PROGRAM Callblocks
VAR
	
CC1_Clamp_Unit1_3 : clamp;
CC2_Clamp_Unit2_3 : clamp;
CC3_Clamp_Unit3_3 : clamp;
CC4_Clamp_Unit4_3 : clamp;
CC5_Clamp_Unit5_1 : clamp;
CC6_Clamp_Unit6_1 : clamp;

Temp_bool : BOOL;
Feedback_Unit1  : Feedback_FB;
Feedback_Unit2  : Feedback_FB;
Feedback_Unit3  : Feedback_FB;
Feedback_Unit4  : Feedback_FB;
Feedback_Unit5  : Feedback_FB;
Feedback_Unit6  : Feedback_FB;


Door           : RollerDoor;
Trunion        : Trunion;
TT             : Turntable ;
Robot1         : Weldrobot;
Robot2         : MHrobot;

END_VAR

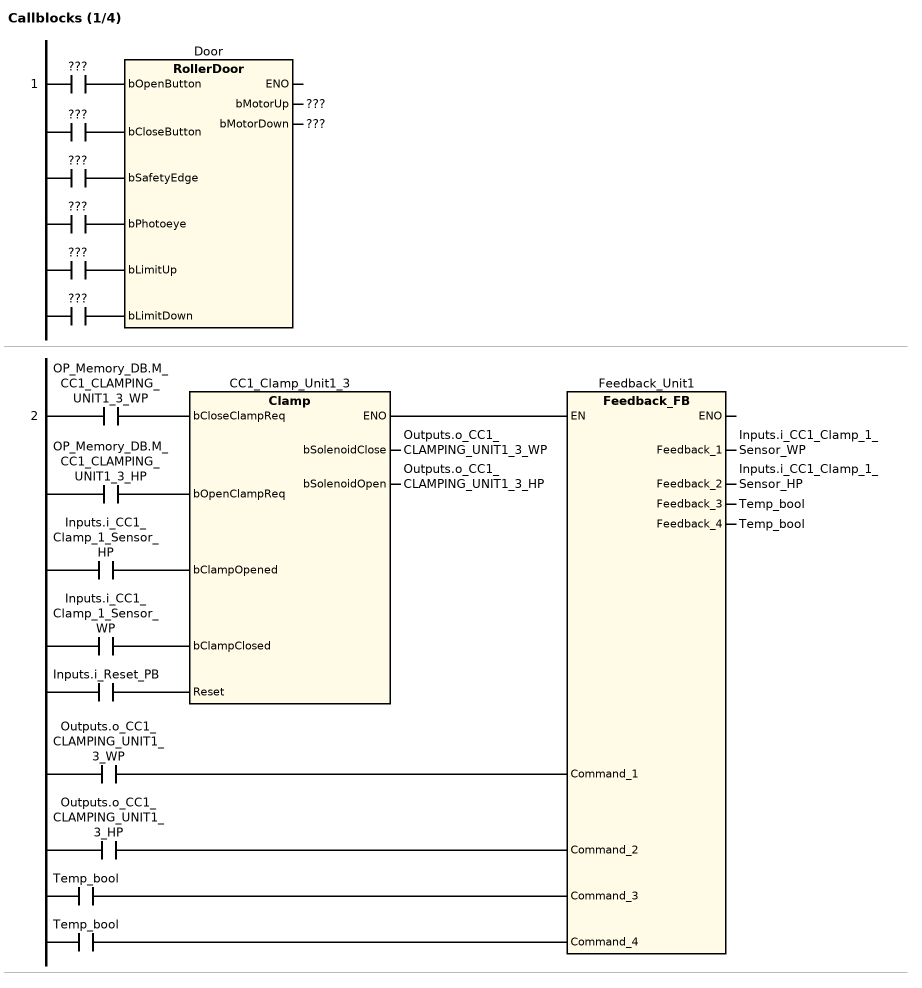
// NETWORK 1
Door(); // RollerDoor

// NETWORK 2
CC1_Clamp_Unit1_3(
    bCloseClampReq := OP_Memory_DB.M_CC1_CLAMPING_UNIT1_3_WP,
    bOpenClampReq := OP_Memory_DB.M_CC1_CLAMPING_UNIT1_3_HP,
    bClampOpened := Inputs.i_CC1_Clamp_1_Sensor_HP,
    bClampClosed := Inputs.i_CC1_Clamp_1_Sensor_WP,
    Reset := Inputs.i_Reset_PB,
    bSolenoidClose => Outputs.o_CC1_CLAMPING_UNIT1_3_WP,
    bSolenoidOpen => Outputs.o_CC1_CLAMPING_UNIT1_3_HP); // Clamp
Feedback_Unit1(
    EN := TRUE,
    Command_1 := Outputs.o_CC1_CLAMPING_UNIT1_3_WP,
    Command_2 := Outputs.o_CC1_CLAMPING_UNIT1_3_HP,
    Command_3 := Temp_bool,
    Command_4 := Temp_bool,
    Feedback_1 => Inputs.i_CC1_Clamp_1_Sensor_WP,
    Feedback_2 => Inputs.i_CC1_Clamp_1_Sensor_HP,
    Feedback_3 => Temp_bool,
    Feedback_4 => Temp_bool); // Feedback_FB

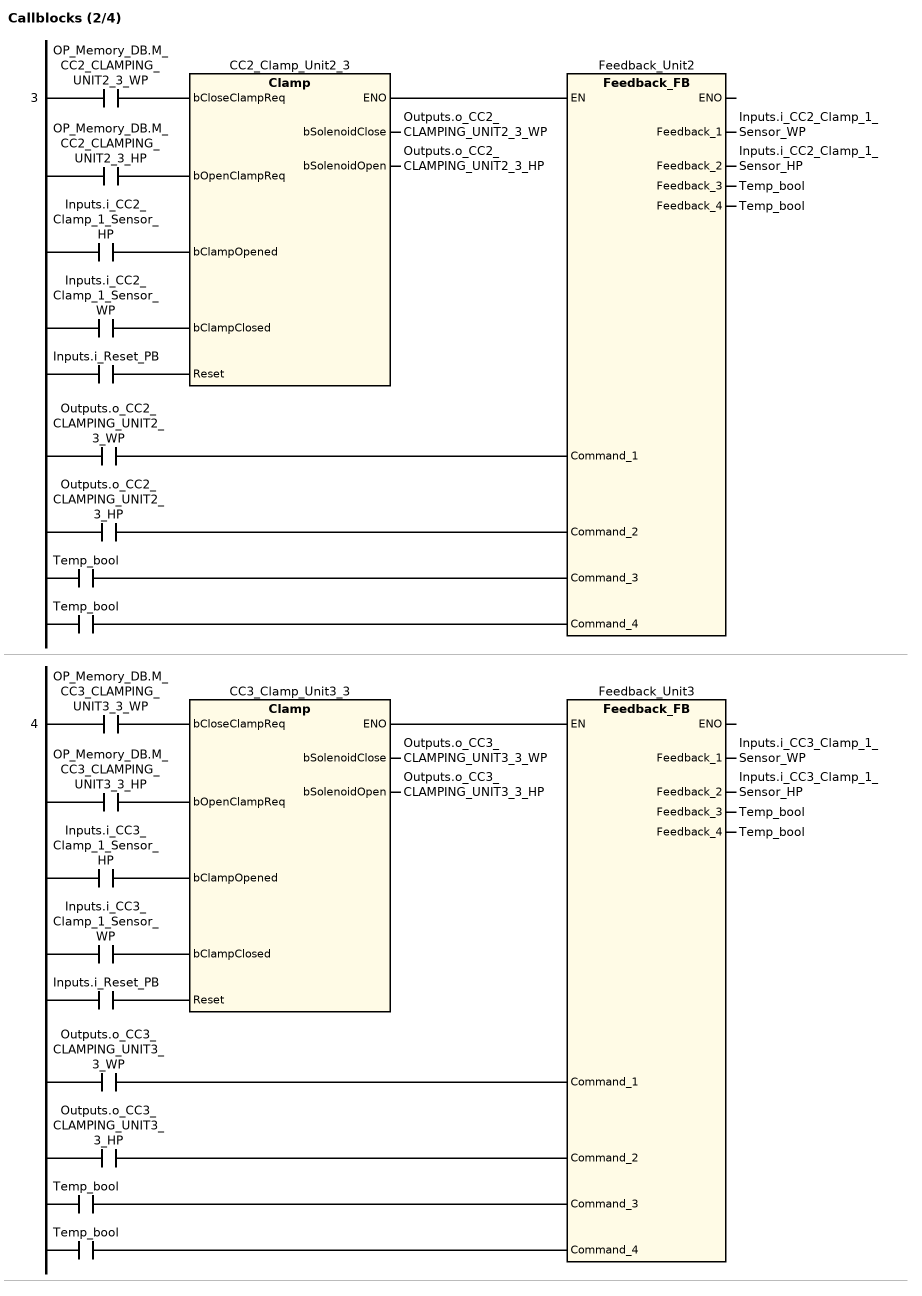
// NETWORK 3
CC2_Clamp_Unit2_3(
    bCloseClampReq := OP_Memory_DB.M_CC2_CLAMPING_UNIT2_3_WP,
    bOpenClampReq := OP_Memory_DB.M_CC2_CLAMPING_UNIT2_3_HP,
    bClampOpened := Inputs.i_CC2_Clamp_1_Sensor_HP,
    bClampClosed := Inputs.i_CC2_Clamp_1_Sensor_WP,
    Reset := Inputs.i_Reset_PB,
    bSolenoidClose => Outputs.o_CC2_CLAMPING_UNIT2_3_WP,
    bSolenoidOpen => Outputs.o_CC2_CLAMPING_UNIT2_3_HP); // Clamp
Feedback_Unit2(
    EN := TRUE,
    Command_1 := Outputs.o_CC2_CLAMPING_UNIT2_3_WP,
    Command_2 := Outputs.o_CC2_CLAMPING_UNIT2_3_HP,
    Command_3 := Temp_bool,
    Command_4 := Temp_bool,
    Feedback_1 => Inputs.i_CC2_Clamp_1_Sensor_WP,
    Feedback_2 => Inputs.i_CC2_Clamp_1_Sensor_HP,
    Feedback_3 => Temp_bool,
    Feedback_4 => Temp_bool); // Feedback_FB

// NETWORK 4
CC3_Clamp_Unit3_3(
    bCloseClampReq := OP_Memory_DB.M_CC3_CLAMPING_UNIT3_3_WP,
    bOpenClampReq := OP_Memory_DB.M_CC3_CLAMPING_UNIT3_3_HP,
    bClampOpened := Inputs.i_CC3_Clamp_1_Sensor_HP,
    bClampClosed := Inputs.i_CC3_Clamp_1_Sensor_WP,
    Reset := Inputs.i_Reset_PB,
    bSolenoidClose => Outputs.o_CC3_CLAMPING_UNIT3_3_WP,
    bSolenoidOpen => Outputs.o_CC3_CLAMPING_UNIT3_3_HP); // Clamp
Feedback_Unit3(
    EN := TRUE,
    Command_1 := Outputs.o_CC3_CLAMPING_UNIT3_3_WP,
    Command_2 := Outputs.o_CC3_CLAMPING_UNIT3_3_HP,
    Command_3 := Temp_bool,
    Command_4 := Temp_bool,
    Feedback_1 => Inputs.i_CC3_Clamp_1_Sensor_WP,
    Feedback_2 => Inputs.i_CC3_Clamp_1_Sensor_HP,
    Feedback_3 => Temp_bool,
    Feedback_4 => Temp_bool); // Feedback_FB

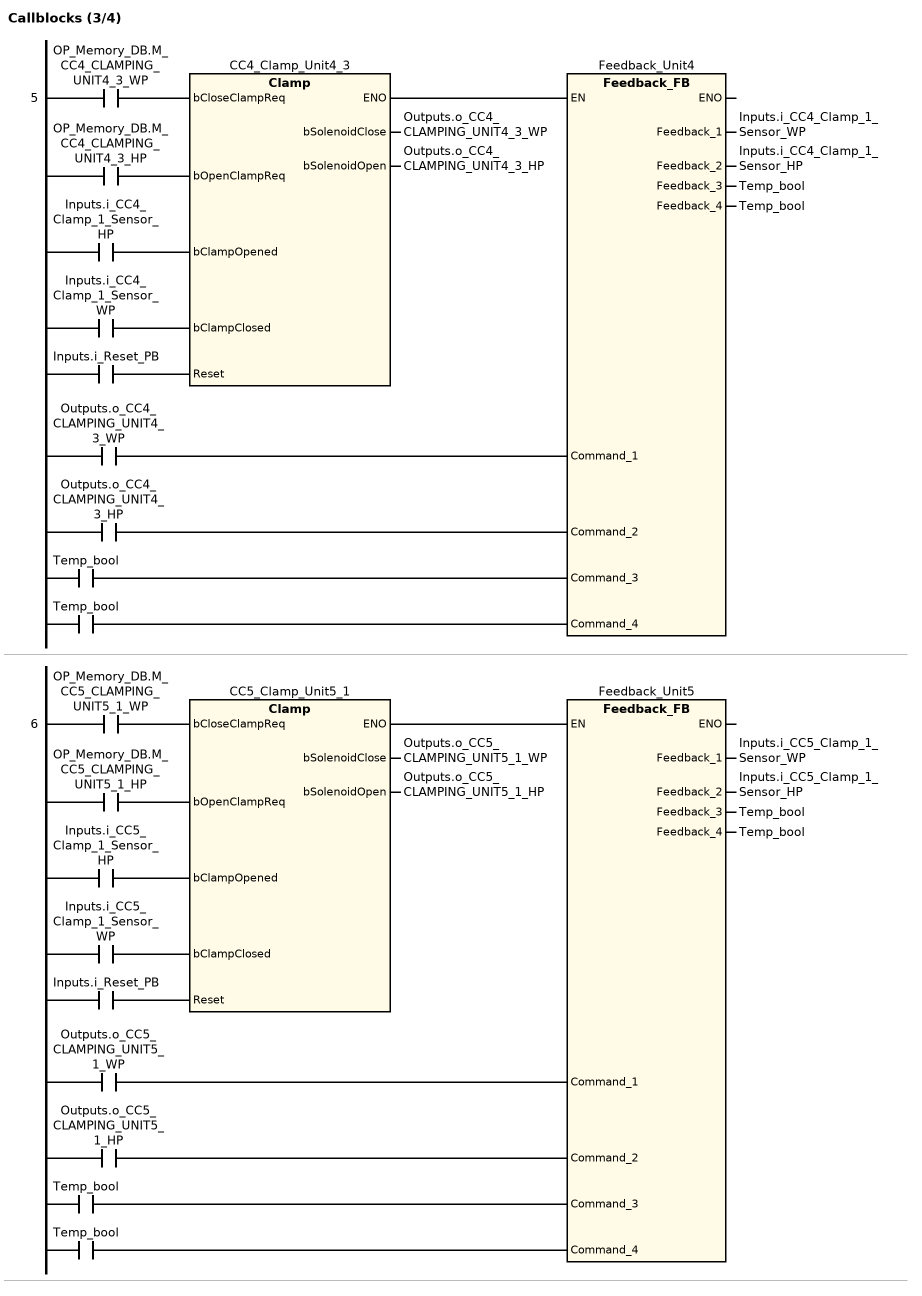
// NETWORK 5
CC4_Clamp_Unit4_3(
    bCloseClampReq := OP_Memory_DB.M_CC4_CLAMPING_UNIT4_3_WP,
    bOpenClampReq := OP_Memory_DB.M_CC4_CLAMPING_UNIT4_3_HP,
    bClampOpened := Inputs.i_CC4_Clamp_1_Sensor_HP,
    bClampClosed := Inputs.i_CC4_Clamp_1_Sensor_WP,
    Reset := Inputs.i_Reset_PB,
    bSolenoidClose => Outputs.o_CC4_CLAMPING_UNIT4_3_WP,
    bSolenoidOpen => Outputs.o_CC4_CLAMPING_UNIT4_3_HP); // Clamp
Feedback_Unit4(
    EN := TRUE,
    Command_1 := Outputs.o_CC4_CLAMPING_UNIT4_3_WP,
    Command_2 := Outputs.o_CC4_CLAMPING_UNIT4_3_HP,
    Command_3 := Temp_bool,
    Command_4 := Temp_bool,
    Feedback_1 => Inputs.i_CC4_Clamp_1_Sensor_WP,
    Feedback_2 => Inputs.i_CC4_Clamp_1_Sensor_HP,
    Feedback_3 => Temp_bool,
    Feedback_4 => Temp_bool); // Feedback_FB

// NETWORK 6
CC5_Clamp_Unit5_1(
    bCloseClampReq := OP_Memory_DB.M_CC5_CLAMPING_UNIT5_1_WP,
    bOpenClampReq := OP_Memory_DB.M_CC5_CLAMPING_UNIT5_1_HP,
    bClampOpened := Inputs.i_CC5_Clamp_1_Sensor_HP,
    bClampClosed := Inputs.i_CC5_Clamp_1_Sensor_WP,
    Reset := Inputs.i_Reset_PB,
    bSolenoidClose => Outputs.o_CC5_CLAMPING_UNIT5_1_WP,
    bSolenoidOpen => Outputs.o_CC5_CLAMPING_UNIT5_1_HP); // Clamp
Feedback_Unit5(
    EN := TRUE,
    Command_1 := Outputs.o_CC5_CLAMPING_UNIT5_1_WP,
    Command_2 := Outputs.o_CC5_CLAMPING_UNIT5_1_HP,
    Command_3 := Temp_bool,
    Command_4 := Temp_bool,
    Feedback_1 => Inputs.i_CC5_Clamp_1_Sensor_WP,
    Feedback_2 => Inputs.i_CC5_Clamp_1_Sensor_HP,
    Feedback_3 => Temp_bool,
    Feedback_4 => Temp_bool); // Feedback_FB

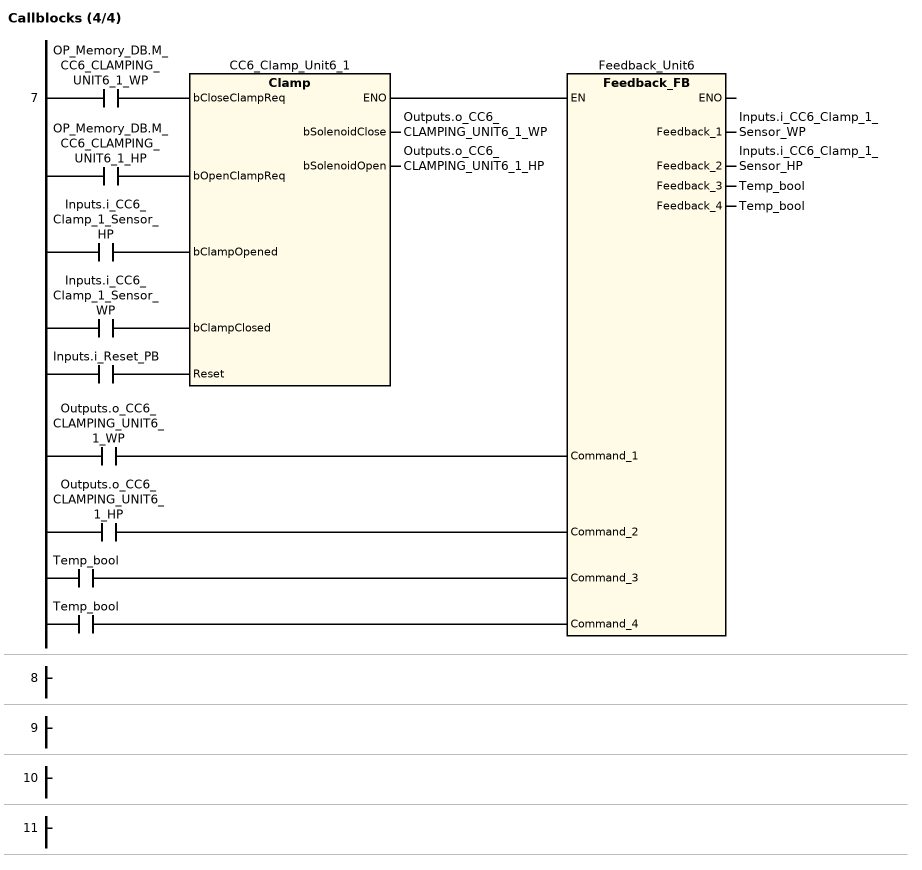
// NETWORK 7
CC6_Clamp_Unit6_1(
    bCloseClampReq := OP_Memory_DB.M_CC6_CLAMPING_UNIT6_1_WP,
    bOpenClampReq := OP_Memory_DB.M_CC6_CLAMPING_UNIT6_1_HP,
    bClampOpened := Inputs.i_CC6_Clamp_1_Sensor_HP,
    bClampClosed := Inputs.i_CC6_Clamp_1_Sensor_WP,
    Reset := Inputs.i_Reset_PB,
    bSolenoidClose => Outputs.o_CC6_CLAMPING_UNIT6_1_WP,
    bSolenoidOpen => Outputs.o_CC6_CLAMPING_UNIT6_1_HP); // Clamp
Feedback_Unit6(
    EN := TRUE,
    Command_1 := Outputs.o_CC6_CLAMPING_UNIT6_1_WP,
    Command_2 := Outputs.o_CC6_CLAMPING_UNIT6_1_HP,
    Command_3 := Temp_bool,
    Command_4 := Temp_bool,
    Feedback_1 => Inputs.i_CC6_Clamp_1_Sensor_WP,
    Feedback_2 => Inputs.i_CC6_Clamp_1_Sensor_HP,
    Feedback_3 => Temp_bool,
    Feedback_4 => Temp_bool); // Feedback_FB

// NETWORK 8

// NETWORK 9

// NETWORK 10

// NETWORK 11

END_PROGRAM

(* stored: Version 1.1.0.1, ProductVersion 3.1.4024.16
   POU Callblocks: Id {75f125e3-d2f9-4c45-a66e-fca76e6d708f}, SpecialFunc None *)
